// TwinCAT 3 PLC project CycleManagerInterfaceLib
// Title: CNM_CycleManagerInterfaces
// Company: ekvip automation GmbH
// Author: tdie
// ProjectVersion: 0.1.1.0
// Description: A library to provide interfaces and the API for Cycle Managing. .. <legal notes> legal notes ================= | SPDX-FileCopyrightText: © 2024 ekvip automation GmbH <info@ekvip.de> | SPDX-License-Identifier: Apache-2.0 | For details check: Apache-2.0_ .. _Apache-2.0: https://www.apache.org/licenses/LICENSE-2.0 .. </legal notes>
// ProgramVersion: 3.1.4026.19
// libraries:
//   CNM_AbstractObject, * (ekvip automation GmbH)
//   CNM_AssertionInterfaces, * (ekvip automation GmbH)
//   CNM_CommandInterfaces, * (ekvip automation GmbH)
//   CNM_MessageInterfaces, * (ekvip automation GmbH)
//   CNM_ReturnTypes, * (ekvip automation GmbH)
//   Tc2_Standard, * (Beckhoff Automation GmbH)
// project tree:
//   CycleManager/interfaces/configuration/ ICycleManagerConfiguration.TcIO, ICycleManagerConfigurationScope.TcIO, ICycleManagerDefaultParameters.TcIO, ICycleManagerParameters.TcIO, IPauseConfiguration.TcIO, IStopRequestConfiguration.TcIO, ISteppingConfiguration.TcIO, ISequenceConfiguration.TcIO, IStepConfiguration.TcIO, StepStopRequestMode.TcDUT
//   CycleManager/interfaces/ ICycleError.TcIO, ICycleSteps.TcIO
//   CycleManager/SingleExecution/interfaces/ ISingleExecutionCycleManager.TcIO
//   Project Information/ F_GetCompany.TcPOU, F_GetTitle.TcPOU, F_GetVersion.TcPOU
//   Version/ Global_Version.TcGVL
// real-time tasks:
//   TASK PlcTask: cycle T#10ms, priority 20, ADS port 350

// ---- CycleManager/interfaces/configuration/StepStopRequestMode.TcDUT
(*

## Short summary
``StepStopRequestMode`` is an enumeration to control StopRequest behaviour in cycle managers.
Cycle managers should continue with SUCCESS after a stop request is acknowledged by the cycle manager.

.. <legal notes>

legal notes
=================
| SPDX-FileCopyrightText: © 2024 ekvip automation GmbH <info@ekvip.de>
| SPDX-License-Identifier: Apache-2.0
| For details check: Apache-2.0_

.. _Apache-2.0: https://www.apache.org/licenses/LICENSE-2.0

.. </legal notes>

enumeration values
======================

*)

{attribute 'qualified_only'}
{attribute 'strict'}
{attribute 'to_string'}
TYPE StepStopRequestMode :
(
	(*ignore stop request*)
	IGNORE := 0,
	(*proceed with stop request after step finishes and would proceed*)
	AFTER_SUCCESSFUL_STEP := 1,
	(*proceed with stop request only if the step is still busy*)
	ON_BUSY := 2,
	(*immediately proceed with stop request*)
	IMMEDIATE := 3
)DINT;
END_TYPE

// ---- Version/Global_Version.TcGVL
{attribute 'TcGenerated'}
{attribute 'no-analysis'}
{attribute 'linkalways'}
// This function has been automatically generated from the project information.
VAR_GLOBAL CONSTANT
	{attribute 'const_non_replaced'}
	stLibVersion_CNM_CycleManagerInterfaces : ST_LibVersion := (iMajor := 0, iMinor := 1, iBuild := 1, iRevision := 0, nFlags := 0, sVersion := '0.1.1.0');
END_VAR

// ---- CycleManager/interfaces/configuration/ICycleManagerConfiguration.TcIO
(*

## Short summary
An interface to provide configurations for cycle manager in a fluent way.

.. <legal notes>

legal notes
=================
| SPDX-FileCopyrightText: © 2024 ekvip automation GmbH <info@ekvip.de>
| SPDX-License-Identifier: Apache-2.0
| For details check: Apache-2.0_

.. _Apache-2.0: https://www.apache.org/licenses/LICENSE-2.0

.. </legal notes>



*)
INTERFACE ICycleManagerConfiguration EXTENDS __SYSTEM.IQueryInterface

(*

## Short summary
An interface to provide configurations for cycle manager in a fluent way.

.. <legal notes>

legal notes
=================
| SPDX-FileCopyrightText: © 2024 ekvip automation GmbH <info@ekvip.de>
| SPDX-License-Identifier: Apache-2.0
| For details check: Apache-2.0_

.. _Apache-2.0: https://www.apache.org/licenses/LICENSE-2.0

.. </legal notes>



*)
PROPERTY configuration : ICycleManagerConfigurationScope
GET
END_GET
END_PROPERTY

END_INTERFACE

// ---- CycleManager/interfaces/configuration/ICycleManagerConfigurationScope.TcIO
(*

## Short summary
An interface to provide a scope selector for configurations in cycle managers.

.. <legal notes>

legal notes
=================
| SPDX-FileCopyrightText: © 2024 ekvip automation GmbH <info@ekvip.de>
| SPDX-License-Identifier: Apache-2.0
| For details check: Apache-2.0_

.. _Apache-2.0: https://www.apache.org/licenses/LICENSE-2.0

.. </legal notes>



*)
INTERFACE ICycleManagerConfigurationScope EXTENDS __SYSTEM.IQueryInterface

PROPERTY sequence : ISequenceConfiguration
GET
END_GET
END_PROPERTY

PROPERTY step : IStepConfiguration
GET
END_GET
END_PROPERTY

END_INTERFACE

// ---- CycleManager/interfaces/configuration/ICycleManagerDefaultParameters.TcIO
(*

## Short summary
An interface to provide configurations for cycle manager default parameters.
Used internally to allow better fluent implementation.

.. <legal notes>

legal notes
=================
| SPDX-FileCopyrightText: © 2024 ekvip automation GmbH <info@ekvip.de>
| SPDX-License-Identifier: Apache-2.0
| For details check: Apache-2.0_

.. _Apache-2.0: https://www.apache.org/licenses/LICENSE-2.0

.. </legal notes>



*)
INTERFACE ICycleManagerDefaultParameters EXTENDS __System.IQueryInterface

(*

## Short summary
This property sets the default error step for all cycle manager operations.

.. <legal notes>

legal notes
=================
| SPDX-FileCopyrightText: © 2024 ekvip automation GmbH <info@ekvip.de>
| SPDX-License-Identifier: Apache-2.0
| For details check: Apache-2.0_

.. _Apache-2.0: https://www.apache.org/licenses/LICENSE-2.0

.. </legal notes>

*)

PROPERTY defaultErrorStep : DINT
SET
END_SET
END_PROPERTY

(*

## Short summary
This property sets the default pause behavior for all cycle manager operations.

### Usage
This property configures whether pause functionality is enabled by default for the cycle manager.
When enabled, the cycle manager will respond to pause signals and can suspend execution at
appropriate points in the sequence.

The property is write-only and accepts a boolean value to enable or disable pausing.

#### typical usage patterns
1. **Production mode setup**: Enable pausing for production sequences
2. **Maintenance configuration**: Enable pausing for maintenance operations
3. **Automatic operation**: Disable pausing for fully automatic sequences
4. **Operator control**: Enable pausing to allow operator intervention

#### when to use
- During cycle manager initialization to set pause behavior
- When configuring operation modes (automatic vs. manual)
- For setting up operator control capabilities
- When implementing safety or emergency stop procedures

#### behavior details

- When enabled: Cycle manager responds to pause input signals
- When disabled: Pause signals are ignored and sequence continues
- Affects all steps in the sequence unless overridden locally
- Can be overridden on a per-step basis using step configuration

**Example:**
```
// Enable pause for production mode
cyclemanager.configuration.sequence.defaultPauseEnabled := TRUE;

// Disable pause for automatic operation
cyclemanager.configuration.sequence.defaultPauseEnabled := FALSE;

// Configuration based on operation mode
IF operation_mode = OperationMode.MANUAL THEN
	cyclemanager.configuration.sequence.defaultPauseEnabled := TRUE;
ELSE
	cyclemanager.configuration.sequence.defaultPauseEnabled := FALSE;
END_IF;

// Safety configuration
cyclemanager.configuration.sequence
	.defaultPauseEnabled := enable_safety_pause;
```

.. <legal notes>

legal notes
=================
| SPDX-FileCopyrightText: © 2024 ekvip automation GmbH <info@ekvip.de>
| SPDX-License-Identifier: Apache-2.0
| For details check: Apache-2.0_

.. _Apache-2.0: https://www.apache.org/licenses/LICENSE-2.0

.. </legal notes>

*)
PROPERTY defaultPauseEnabled : BOOL
SET
END_SET
END_PROPERTY

(*

## Short summary
Specifies whether the SUCCESS step of the state machine can be skipped when the transition condition to SUCCESS is already fulfilled.

When set to false, the state machine immediately returns SUCCESS as soon as the transition condition to the SUCCESS state is met, 
without executing the dedicated SUCCESS step. This optimization can save one execution cycle per state machine invocation, which is 
especially beneficial in nested or complex state machine structures.

When set to true, the SUCCESS step will always be executed at least once before the state machine returns SUCCESS. This is required 
in cases where the SUCCESS step performs essential actions (e.g., resetting outputs, logging, or cleanup).

The default value is false.

### Use Case:
Use false when the SUCCESS step has no functional side effects and skipping it can improve performance.
Use true when the SUCCESS step contains logic that must be executed explicitly.

.. <legal notes>

legal notes
=================
| SPDX-FileCopyrightText: © 2025 ekvip automation GmbH <info@ekvip.de>
| SPDX-License-Identifier: Apache-2.0
| For details check: Apache-2.0_

.. _Apache-2.0: https://www.apache.org/licenses/LICENSE-2.0

.. </legal notes>

*)

PROPERTY defaultRequireSuccessStep : BOOL
SET
END_SET
END_PROPERTY

(*

## Short summary
This property sets the default stepping mode configuration after a step change.

.. <legal notes>

legal notes
=================
| SPDX-FileCopyrightText: © 2024 ekvip automation GmbH <info@ekvip.de>
| SPDX-License-Identifier: Apache-2.0
| For details check: Apache-2.0_

.. _Apache-2.0: https://www.apache.org/licenses/LICENSE-2.0

.. </legal notes>

*)

PROPERTY defaultSteppingEnabled : BOOL
SET
END_SET
END_PROPERTY

(*

## Short summary
This property sets the default the step width.

.. <legal notes>

legal notes
=================
| SPDX-FileCopyrightText: © 2024 ekvip automation GmbH <info@ekvip.de>
| SPDX-License-Identifier: Apache-2.0
| For details check: Apache-2.0_

.. _Apache-2.0: https://www.apache.org/licenses/LICENSE-2.0

.. </legal notes>

*)

PROPERTY defaultStepWidth : DINT
SET
END_SET
END_PROPERTY

(*

## Short summary
This property sets the default step mode configuration. 

.. <legal notes>

legal notes
=================
| SPDX-FileCopyrightText: © 2024 ekvip automation GmbH <info@ekvip.de>
| SPDX-License-Identifier: Apache-2.0
| For details check: Apache-2.0_

.. _Apache-2.0: https://www.apache.org/licenses/LICENSE-2.0

.. </legal notes>

*)

PROPERTY defaultStopRequestMode :StepStopRequestMode
SET
END_SET
END_PROPERTY

(*

## Short summary
This property sets the maximum execution time for steps. 
The cycle manager will go into the timeoutStep after the time elapsed.

.. <legal notes>

legal notes
=================
| SPDX-FileCopyrightText: © 2024 ekvip automation GmbH <info@ekvip.de>
| SPDX-License-Identifier: Apache-2.0
| For details check: Apache-2.0_

.. _Apache-2.0: https://www.apache.org/licenses/LICENSE-2.0

.. </legal notes>

*)

PROPERTY defaultTimeout : TIME
SET
END_SET
END_PROPERTY

(*

## Short summary
This property sets the default step that will be set if the current step reaches a timeout. 

.. <legal notes>

legal notes
=================
| SPDX-FileCopyrightText: © 2024 ekvip automation GmbH <info@ekvip.de>
| SPDX-License-Identifier: Apache-2.0
| For details check: Apache-2.0_

.. _Apache-2.0: https://www.apache.org/licenses/LICENSE-2.0

.. </legal notes>

*)

PROPERTY defaultTimeoutStep : DINT
SET
END_SET
END_PROPERTY

END_INTERFACE

// ---- CycleManager/interfaces/configuration/ICycleManagerParameters.TcIO
(*

## Short summary
An interface to provide configurations for the cycle manager parameters.

.. <legal notes>

legal notes
=================
| SPDX-FileCopyrightText: © 2024 ekvip automation GmbH <info@ekvip.de>
| SPDX-License-Identifier: Apache-2.0
| For details check: Apache-2.0_

.. _Apache-2.0: https://www.apache.org/licenses/LICENSE-2.0

.. </legal notes>



*)
INTERFACE ICycleManagerParameters EXTENDS __System.IQueryInterface

(*

## Short summary
This property sets the next step in case of an error.

.. <legal notes>

legal notes
=================
| SPDX-FileCopyrightText: © 2024 ekvip automation GmbH <info@ekvip.de>
| SPDX-License-Identifier: Apache-2.0
| For details check: Apache-2.0_

.. _Apache-2.0: https://www.apache.org/licenses/LICENSE-2.0

.. </legal notes>

*)
PROPERTY errorStep :DINT
SET
END_SET
END_PROPERTY

(*

## Short summary
This property allows enabling and disabling pausing.

.. <legal notes>

legal notes
=================
| SPDX-FileCopyrightText: © 2024 ekvip automation GmbH <info@ekvip.de>
| SPDX-License-Identifier: Apache-2.0
| For details check: Apache-2.0_

.. _Apache-2.0: https://www.apache.org/licenses/LICENSE-2.0

.. </legal notes>

*)

PROPERTY pause : IPauseConfiguration
GET
END_GET
END_PROPERTY

(*

## Short summary
This property allows enabling and disabling stepping mode.

.. <legal notes>

legal notes
=================
| SPDX-FileCopyrightText: © 2024 ekvip automation GmbH <info@ekvip.de>
| SPDX-License-Identifier: Apache-2.0
| For details check: Apache-2.0_

.. _Apache-2.0: https://www.apache.org/licenses/LICENSE-2.0

.. </legal notes>

*)

PROPERTY stepping : ISteppingConfiguration
GET
END_GET
END_PROPERTY

(*

## Short summary
This property sets the step width when proceeding automatically.
This defaults to 1.

.. <legal notes>

legal notes
=================
| SPDX-FileCopyrightText: © 2024 ekvip automation GmbH <info@ekvip.de>
| SPDX-License-Identifier: Apache-2.0
| For details check: Apache-2.0_

.. _Apache-2.0: https://www.apache.org/licenses/LICENSE-2.0

.. </legal notes>

*)
PROPERTY stepWidth : DINT
SET
END_SET
END_PROPERTY

(*

## Short summary
This property allows changing the stop request behaviour in case of active stop request.

.. <legal notes>

legal notes
=================
| SPDX-FileCopyrightText: © 2024 ekvip automation GmbH <info@ekvip.de>
| SPDX-License-Identifier: Apache-2.0
| For details check: Apache-2.0_

.. _Apache-2.0: https://www.apache.org/licenses/LICENSE-2.0

.. </legal notes>

*)
PROPERTY stopRequest : IStopRequestConfiguration
GET
END_GET
END_PROPERTY

(*

## Short summary
This property sets the maximum execution time for steps. 
The cycle manager will go into the timeoutStep after the time elapsed.
Set to T#0MS for no timeout (infinite), default.

.. <legal notes>

legal notes
=================
| SPDX-FileCopyrightText: © 2024 ekvip automation GmbH <info@ekvip.de>
| SPDX-License-Identifier: Apache-2.0
| For details check: Apache-2.0_

.. _Apache-2.0: https://www.apache.org/licenses/LICENSE-2.0

.. </legal notes>

*)
PROPERTY timeout :TIME
SET
END_SET
END_PROPERTY

(*

## Short summary
This property sets the step that will be set if the current step reaches a timeout. 
If not changed will default to the current errorStep.

.. <legal notes>

legal notes
=================
| SPDX-FileCopyrightText: © 2024 ekvip automation GmbH <info@ekvip.de>
| SPDX-License-Identifier: Apache-2.0
| For details check: Apache-2.0_

.. _Apache-2.0: https://www.apache.org/licenses/LICENSE-2.0

.. </legal notes>

*)
PROPERTY timeoutStep :DINT
SET
END_SET
END_PROPERTY

END_INTERFACE

// ---- CycleManager/interfaces/configuration/IPauseConfiguration.TcIO
(*

## Short summary
An interface to enable and diable pause functionallity.

.. <legal notes>

legal notes
=================
| SPDX-FileCopyrightText: © 2024 ekvip automation GmbH <info@ekvip.de>
| SPDX-License-Identifier: Apache-2.0
| For details check: Apache-2.0_

.. _Apache-2.0: https://www.apache.org/licenses/LICENSE-2.0

.. </legal notes>



*)
INTERFACE IPauseConfiguration EXTENDS __System.IQueryInterface

(*

## Short summary
This method disables pausing, disabling the cycle manager transition to PAUSED even if pause signal is active.

.. <legal notes>

legal notes
=================
| SPDX-FileCopyrightText: © 2024 ekvip automation GmbH <info@ekvip.de>
| SPDX-License-Identifier: Apache-2.0
| For details check: Apache-2.0_

.. _Apache-2.0: https://www.apache.org/licenses/LICENSE-2.0

.. </legal notes>

*)
METHOD disable
END_METHOD

(*

## Short summary
This method enables pausing, allowing the cycle manager to transition to PAUSED state if pause is active.

.. <legal notes>

legal notes
=================
| SPDX-FileCopyrightText: © 2024 ekvip automation GmbH <info@ekvip.de>
| SPDX-License-Identifier: Apache-2.0
| For details check: Apache-2.0_

.. _Apache-2.0: https://www.apache.org/licenses/LICENSE-2.0

.. </legal notes>

*)

METHOD enable
END_METHOD

END_INTERFACE

// ---- CycleManager/interfaces/configuration/IStopRequestConfiguration.TcIO
(*

## Short summary
An interface to configure stop request behavior.

.. <legal notes>

legal notes
=================
| SPDX-FileCopyrightText: © 2024 ekvip automation GmbH <info@ekvip.de>
| SPDX-License-Identifier: Apache-2.0
| For details check: Apache-2.0_

.. _Apache-2.0: https://www.apache.org/licenses/LICENSE-2.0

.. </legal notes>



*)
INTERFACE IStopRequestConfiguration EXTENDS __System.IQueryInterface

(*

## Short summary
This method sets the stop request behaviour to ``StepStopRequestMode.AFTER_SUCCESSFUL_STEP``.
If the StopRequest signal is active, the cycle manager will move to succees if the current step was successful during the update call.

.. <legal notes>

legal notes
=================
| SPDX-FileCopyrightText: © 2024 ekvip automation GmbH <info@ekvip.de>
| SPDX-License-Identifier: Apache-2.0
| For details check: Apache-2.0_

.. _Apache-2.0: https://www.apache.org/licenses/LICENSE-2.0

.. </legal notes>


*)

METHOD afterSuccessfulStep
END_METHOD

(*

## Short summary
This method sets the stop request behaviour to ``StepStopRequestMode.IGNORE``.
The cycle manager will ignore the stop request signal.

.. <legal notes>

legal notes
=================
| SPDX-FileCopyrightText: © 2024 ekvip automation GmbH <info@ekvip.de>
| SPDX-License-Identifier: Apache-2.0
| For details check: Apache-2.0_

.. _Apache-2.0: https://www.apache.org/licenses/LICENSE-2.0

.. </legal notes>


*)

METHOD ignore
END_METHOD

(*

## Short summary
This method sets the stop request behaviour to ``StepStopRequestMode.IMMEDIATE``.
If the StopRequest signal is active, the cycle manager will always move to succees during the update call.

.. <legal notes>

legal notes
=================
| SPDX-FileCopyrightText: © 2024 ekvip automation GmbH <info@ekvip.de>
| SPDX-License-Identifier: Apache-2.0
| For details check: Apache-2.0_

.. _Apache-2.0: https://www.apache.org/licenses/LICENSE-2.0

.. </legal notes>


*)

METHOD immediate
END_METHOD

(*

## Short summary
This method sets the stop request behaviour to ``StepStopRequestMode.ON_BUSY``.
If the StopRequest signal is active, the cycle manager will move to succees if the current step was busy during the update call.

.. <legal notes>

legal notes
=================
| SPDX-FileCopyrightText: © 2024 ekvip automation GmbH <info@ekvip.de>
| SPDX-License-Identifier: Apache-2.0
| For details check: Apache-2.0_

.. _Apache-2.0: https://www.apache.org/licenses/LICENSE-2.0

.. </legal notes>

*)

METHOD onBusy
END_METHOD

END_INTERFACE

// ---- CycleManager/interfaces/configuration/ISteppingConfiguration.TcIO
(*

## Short summary
An interface to provide stepping behaviour to cycle managers.

.. <legal notes>

legal notes
=================
| SPDX-FileCopyrightText: © 2024 ekvip automation GmbH <info@ekvip.de>
| SPDX-License-Identifier: Apache-2.0
| For details check: Apache-2.0_

.. _Apache-2.0: https://www.apache.org/licenses/LICENSE-2.0

.. </legal notes>



*)
INTERFACE ISteppingConfiguration EXTENDS __System.IQueryInterface

(*

## Short summary
This method disables step mode, allowing automatic proceeding without using the step signal.

.. <legal notes>

legal notes
=================
| SPDX-FileCopyrightText: © 2024 ekvip automation GmbH <info@ekvip.de>
| SPDX-License-Identifier: Apache-2.0
| For details check: Apache-2.0_

.. _Apache-2.0: https://www.apache.org/licenses/LICENSE-2.0

.. </legal notes>

*)
METHOD disable
END_METHOD

(*

## Short summary
This method enables step mode, only allowing automatic proceeding if the step signal is active.

.. <legal notes>

legal notes
=================
| SPDX-FileCopyrightText: © 2024 ekvip automation GmbH <info@ekvip.de>
| SPDX-License-Identifier: Apache-2.0
| For details check: Apache-2.0_

.. _Apache-2.0: https://www.apache.org/licenses/LICENSE-2.0

.. </legal notes>

*)
METHOD enable
END_METHOD

END_INTERFACE

// ---- CycleManager/interfaces/configuration/ISequenceConfiguration.TcIO
(*

## Short summary
An interface to provide configurations for all cycle manager steps.
Should affect the all steps in the cycle manager (default values).

.. <legal notes>

legal notes
=================
| SPDX-FileCopyrightText: © 2024 ekvip automation GmbH <info@ekvip.de>
| SPDX-License-Identifier: Apache-2.0
| For details check: Apache-2.0_

.. _Apache-2.0: https://www.apache.org/licenses/LICENSE-2.0

.. </legal notes>



*)
INTERFACE ISequenceConfiguration EXTENDS ICycleManagerParameters

(*

## Short summary
Specifies whether the SUCCESS step of the state machine can be skipped when the transition condition to SUCCESS is already fulfilled.

When set to false, the state machine immediately returns SUCCESS as soon as the transition condition to the SUCCESS state is met, 
without executing the dedicated SUCCESS step. This optimization can save one execution cycle per state machine invocation, which is 
especially beneficial in nested or complex state machine structures.

When set to true, the SUCCESS step will always be executed at least once before the state machine returns SUCCESS. This is required 
in cases where the SUCCESS step performs essential actions (e.g., resetting outputs, logging, or cleanup).

The default value is false.

### Use Case
Use false when the SUCCESS step has no functional side effects and skipping it can improve performance.
Use true when the SUCCESS step contains logic that must be executed explicitly.

.. <legal notes>

legal notes
=================
| SPDX-FileCopyrightText: © 2025 ekvip automation GmbH <info@ekvip.de>
| SPDX-License-Identifier: Apache-2.0
| For details check: Apache-2.0_

.. _Apache-2.0: https://www.apache.org/licenses/LICENSE-2.0

.. </legal notes>

*)

PROPERTY requireSuccessStep : BOOL
SET
END_SET
END_PROPERTY

END_INTERFACE

// ---- CycleManager/interfaces/configuration/IStepConfiguration.TcIO
(*

## Short summary
An interface to provide configurations for cycle manager steps.
Should only affect the currently active step.

.. <legal notes>

legal notes
=================
| SPDX-FileCopyrightText: © 2024 ekvip automation GmbH <info@ekvip.de>
| SPDX-License-Identifier: Apache-2.0
| For details check: Apache-2.0_

.. _Apache-2.0: https://www.apache.org/licenses/LICENSE-2.0

.. </legal notes>



*)
INTERFACE IStepConfiguration EXTENDS ICycleManagerParameters

END_INTERFACE

// ---- CycleManager/interfaces/ICycleError.TcIO
(*

## Short summary
An interface to provide error handling in cycle management.

.. <legal notes>

legal notes
=================
| SPDX-FileCopyrightText: © 2024 ekvip automation GmbH <info@ekvip.de>
| SPDX-License-Identifier: Apache-2.0
| For details check: Apache-2.0_

.. _Apache-2.0: https://www.apache.org/licenses/LICENSE-2.0

.. </legal notes>



*)
INTERFACE ICycleError EXTENDS __System.IQueryInterface

(*

## Short summary
This method acknowledges an error in the cycle manager 
and resets the current step to the step before the error occurred.


### Purpose and usage
This method provides error acknowledgment functionality for the cycle manager. It clears the current error state
and returns the cycle manager to the step that was executing before the error occurred, allowing for error recovery
and continuation of the sequence.

The method should be called when an operator or system wants to acknowledge an error and attempt to continue
the process from where it left off.

### Typical usage patterns

1. **Manual error acknowledgment**: Operator acknowledges error via HMI button
2. **Automatic error recovery**: System automatically acknowledges after conditions are met
3. **Retry operations**: Acknowledge error to retry the failed step
4. **Error logging**: Acknowledge error after logging for audit trail

#### When to use

- When an error has been resolved and process should continue
- After manual operator intervention to fix the error condition
- In automated error recovery scenarios
- When implementing retry logic after temporary failures

### behavior

- Clears the error state flag
- Returns cycle manager to the last successful step
- Resets internal error tracking variables
- Allows normal sequence progression to resume

**Example:**
```
// Manual error acknowledgment via HMI
IF HMI_acknowledge_button THEN
	cyclemanager.errors.acknowledge();
	HMI_acknowledge_button := FALSE;
END_IF;

// Automatic error acknowledgment after condition resolution
ERROR_STEP:
	IF error_condition_resolved THEN
		cyclemanager.errors.acknowledge();  // Return to previous step
	END_IF;

// Error acknowledgment with logging
IF error_acknowledged_by_operator THEN
	logger.logEvent('Error acknowledged by operator');
	cyclemanager.errors.acknowledge();
	error_acknowledged_by_operator := FALSE;
END_IF;
```

.. <legal notes>

legal notes
=================
| SPDX-FileCopyrightText: © 2024 ekvip automation GmbH <info@ekvip.de>
| SPDX-License-Identifier: Apache-2.0
| For details check: Apache-2.0_

.. _Apache-2.0: https://www.apache.org/licenses/LICENSE-2.0

.. </legal notes>

*)
METHOD acknowledge
END_METHOD

(*

## Short summary
This method throws an alarm and waits for it to be confirmed. 
When the alarm was confirmed the cyclemanager will proceed to next configured step.
If the current step is the result of an evaluated error state and the input 'resumeWithLastStep' is set to true, the cyclemanager will proceed to the last step.
**Warning:**  The 'resumeWithLastStep' flag will be ignored if the last step was successful.

### Purpose and usage
This method provides comprehensive error handling by displaying an alarm to the operator and managing 
the subsequent cycle manager behavior based on the error acknowledgment. It integrates alarm management
with cycle flow control for robust error handling.

The method blocks execution until the alarm is acknowledged and then determines the next step based
on the error context and resumeWithLastStep parameter.

### Typical usage patterns
1. **Critical error handling**: Display alarm for critical errors requiring operator intervention
2. **Process deviation handling**: Show alarm when process parameters are out of range
3. **Equipment failure handling**: Alert operators to equipment malfunctions
4. **Recovery operations**: Provide options for continuing after error resolution

### When to use
- When an error requires operator notification and acknowledgment
- For errors that need to be logged and tracked in the alarm system
- When you need flexible recovery options (continue or retry)
- For integrating cycle management with plant-wide alarm systems

### Behaviour details
- Displays the alarm using the CNM message system
- Blocks cycle progression until alarm is acknowledged
- If resumeWithLastStep=TRUE and step was reached via error: returns to last step
- If resumeWithLastStep=FALSE: proceeds to next configured step
- Warning: resumeWithLastStep is ignored if last step was successful

### Parameter validation
- alarm parameter must be a valid IAlarm instance
- resumeWithLastStep flag only affects behavior when current step resulted from error evaluation

**Example:**
```
// Basic error handling with alarm
PROCESS_STEP:
	IF motor_overload_detected THEN
		cyclemanager.errors.handle(motor_overload_alarm, TRUE);  // Resume with last step after ack
	END_IF;

// Error handling with different recovery strategies
CRITICAL_OPERATION:
	IF safety_violation THEN
		cyclemanager.errors.handle(safety_alarm, FALSE);  // Don't resume, go to next step
	ELSIF equipment_fault THEN
		cyclemanager.errors.handle(equipment_alarm, TRUE);  // Allow retry of operation
	END_IF;

// Complex error handling with context
VAR
	process_error_alarm : ProcessErrorAlarm;
END_VAR

MONITORING_STEP:
	IF temperature_out_of_range THEN
		process_error_alarm.setMessage('Temperature exceeded limits');
		process_error_alarm.setSeverity(AlarmSeverity.WARNING);
		cyclemanager.errors.handle(process_error_alarm, TRUE);
	END_IF;
```

.. <legal notes>

legal notes
=================
| SPDX-FileCopyrightText: © 2024 ekvip automation GmbH <info@ekvip.de>
| SPDX-License-Identifier: Apache-2.0
| For details check: Apache-2.0_

.. _Apache-2.0: https://www.apache.org/licenses/LICENSE-2.0

.. </legal notes>

*)

METHOD handle
VAR_INPUT
	(* the alarm event that should be thrown *)
	alarm :CNM_MessageInterfaces.IAlarm;
	(* if this flag is set AND we got to the current step because of an ERROR state, then the cyclemanager will automatically will go back to the last step *)
	resumeWithLastStep :BOOL := TRUE;
END_VAR
END_METHOD

(*

## Short summary
This property returns TRUE if the step was reached by evaluating an error.

### Purpose and usage
This property provides status information about how the current step was reached. It indicates whether 
the cycle manager arrived at the current step as a result of an error evaluation, which is crucial
for implementing context-aware error handling and recovery logic.

The property is read-only and returns a boolean value indicating error context.

**return**
BOOL: TRUE if current step was reached by error evaluation, FALSE if reached through normal flow

### Typical usage patterns
1. **Conditional error handling**: Different behavior based on how step was reached
2. **Recovery decision making**: Determine appropriate recovery actions
3. **Error logging**: Log additional context about error conditions
4. **UI feedback**: Show different information based on error context

### When to use
- In error handling steps to determine recovery strategy
- When implementing different behaviors for error vs. normal flow
- For logging and audit trail purposes
- In HMI displays to show appropriate error context

### Behaviour details
- Returns TRUE when step was reached via error evaluation (e.g., command returned ERROR state)
- Returns FALSE when step was reached through normal progression
- Useful for implementing smart error recovery logic
- Context is maintained until step changes or error is acknowledged

**Example:**
```
// Context-aware error handling
ERROR_STEP:
	IF cyclemanager.errors.isInErrorStep THEN
		// This step was reached due to an error
		display_error_message := 'Process failed - manual intervention required';
		allow_retry := TRUE;
	ELSE
		// This step was reached through normal flow
		display_error_message := 'Manual error step - check process conditions';
		allow_retry := FALSE;
	END_IF;

// Different recovery strategies based on context
RECOVERY_STEP:
	IF cyclemanager.errors.isInErrorStep THEN
		// Automatic retry for error-triggered steps
		IF retry_count < MAX_RETRIES THEN
			cyclemanager.errors.acknowledge();  // Try again
		ELSE
			cyclemanager.steps.next := ABORT_STEP;  // Give up
		END_IF;
	ELSE
		// Manual step - wait for operator decision
		cyclemanager.waitFor(operator_continue_signal);
	END_IF;

// Error logging with context
IF log_step_entry THEN
	IF cyclemanager.errors.isInErrorStep THEN
		logger.logError('Entered step due to error condition');
	ELSE
		logger.logInfo('Entered step through normal flow');
	END_IF;
	log_step_entry := FALSE;
END_IF;

.. <legal notes>

legal notes
=================
| SPDX-FileCopyrightText: © 2024 ekvip automation GmbH <info@ekvip.de>
| SPDX-License-Identifier: Apache-2.0
| For details check: Apache-2.0_

.. _Apache-2.0: https://www.apache.org/licenses/LICENSE-2.0

.. </legal notes>

*)
PROPERTY isInErrorStep : BOOL
GET
END_GET
END_PROPERTY

END_INTERFACE

// ---- CycleManager/interfaces/ICycleSteps.TcIO
(*

## Short summary
An interface to provide last, current and next step properties in cycle management.

.. <legal notes>

legal notes
=================
| SPDX-FileCopyrightText: © 2024 ekvip automation GmbH <info@ekvip.de>
| SPDX-License-Identifier: Apache-2.0
| For details check: Apache-2.0_

.. _Apache-2.0: https://www.apache.org/licenses/LICENSE-2.0

.. </legal notes>



*)
INTERFACE ICycleSteps EXTENDS __System.IQueryInterface

(*

## Short summary
This property returns the current step of the cycle manager.
Proposed use is as CASE control.

### Purpose and usage
This property provides the current step number of the cycle manager for implementing step-based control logic.
It is primarily used in CASE statements to execute different actions based on the current step.

The property is read-only and returns the current step as a DINT value.

**return**
DINT: Current step number of the cycle manager

### Typical usage patterns
1. **CASE control structure**: Main usage in CASE statements for step-based execution
2. **Step monitoring**: Reading current step for HMI display or logging
3. **Conditional logic**: Checking current step for specific conditions

### When to use
- In every cycle manager implementation for step-based control
- When you need to display current step status
- For debugging and logging purposes
- When implementing conditional logic based on current step

**Example:**
```
CASE cyclemanager.steps.current OF
DefaultSteps.STEP.IDLE:
	// Initialize sequence
	;
DefaultSteps.STEP.INIT:
	// Perform initialization
	;
2:
	// Custom step - move to position
	;
3:
	// Custom step - perform operation
	;
4:
	// Custom step - finalize
	;
DefaultSteps.STEP.SUCCESS:
	// Sequence completed successfully
	;
DefaultSteps.STEP.ERROR:
	// Handle error conditions
	;
DefaultSteps.STEP.ABORT:
	// Handle abort conditions
	;
ELSE 
	// Handle unexpected steps
	;
END_CASE

// Usage for monitoring
currentStepForHMI := cyclemanager.steps.current;
```

.. <legal notes>

legal notes
=================
| SPDX-FileCopyrightText: © 2024 ekvip automation GmbH <info@ekvip.de>
| SPDX-License-Identifier: Apache-2.0
| For details check: Apache-2.0_

.. _Apache-2.0: https://www.apache.org/licenses/LICENSE-2.0

.. </legal notes>

*)
PROPERTY current :DINT
GET
END_GET
END_PROPERTY

(*

## Short summary
This property returns the last step of the cycle manager, useful for error steps.

### Purpose and usage
This property provides the last executed step number of the cycle manager, primarily used for error handling and recovery operations.
It allows returning to the previous step for retry operations or error recovery procedures.

The property is read-only and returns the last step as a DINT value.

**return**
DINT: Last executed step number of the cycle manager

### Typical usage patterns
1. **Error recovery**: Returning to previous step after error handling
2. **Retry operations**: Going back one step to retry failed operations
3. **Step debugging**: Tracking step transitions for debugging purposes
4. **Conditional branching**: Making decisions based on where the error occurred

### When to use
- In error handling steps to implement retry logic
- When you need to return to the previous step after error resolution
- For debugging step transitions and sequence flow
- In timeout handling to retry the previous operation

**Example:**
```
// Error handling with retry logic
TIMEOUT_STEP_FOR_RETRY:
	cM.steps.next := cM.steps.last - 1;  // Go back to previous step
	cM.waitFor(ACK);

// Error step with conditional recovery
DefaultSteps.STEP.ERROR:
	IF retry_counter < MAX_RETRIES THEN
		retry_counter := retry_counter + 1;
		cM.steps.next := cM.steps.last;  // Retry the failed step
	ELSE
		cM.steps.next := DefaultSteps.STEP.ABORT;  // Give up after max retries
	END_IF;

// Step transition logging
logger.logStepTransition(cM.steps.last, cM.steps.current);
```

.. <legal notes>

legal notes
=================
| SPDX-FileCopyrightText: © 2024 ekvip automation GmbH <info@ekvip.de>
| SPDX-License-Identifier: Apache-2.0
| For details check: Apache-2.0_

.. _Apache-2.0: https://www.apache.org/licenses/LICENSE-2.0

.. </legal notes>

*)
PROPERTY last :DINT
GET
END_GET
END_PROPERTY

(*

## Short summary
This property sets the next step of the cycle manager.

### Purpose and usage
This property sets the next step that the cycle manager should execute after completing the current step.
It provides explicit control over the sequence flow, allowing for conditional branching, error handling, and custom step sequencing.

The property is write-only and accepts a DINT value representing the target step number.

### Typical usage patterns
1. **Conditional branching**: Setting different next steps based on conditions
2. **Error handling**: Directing flow to error or recovery steps
3. **Sequential control**: Explicitly controlling step progression
4. **Skip operations**: Jumping over steps that are not needed

### When to use
- When you need to control step progression explicitly
- For conditional branching based on process conditions
- In error handling to redirect to error steps
- When implementing complex sequence logic with jumps
- For skipping steps that are not required in current context

### Parameter validation
- Step number should be a valid step in your sequence
- Negative step numbers are typically reserved for system steps
- Use DefaultSteps.STEP constants for standard steps (IDLE, INIT, SUCCESS, ERROR, ABORT)

**Example:**
```
// Conditional branching
MY_STEP:
	IF process_complete THEN
		cyclemanager.steps.next := SUCCESS_STEP;
	ELSE
		cyclemanager.steps.next := CONTINUE_PROCESS_STEP;
	END_IF;
	cyclemanager.executeCommand(finalizeProcess);

// Error handling
PROCESS_STEP:
	IF error_detected THEN
		cyclemanager.steps.next := DefaultSteps.STEP.ERROR;
	ELSE
		cyclemanager.steps.next := NEXT_PROCESS_STEP;
	END_IF;

// Skip operation based on condition
OPTIONAL_STEP_CHECK:
	IF skip_calibration THEN
		cyclemanager.steps.next := MAIN_OPERATION_STEP;  // Skip calibration
	ELSE
		cyclemanager.steps.next := CALIBRATION_STEP;     // Perform calibration
	END_IF;
```

.. <legal notes>

legal notes
=================
| SPDX-FileCopyrightText: © 2024 ekvip automation GmbH <info@ekvip.de>
| SPDX-License-Identifier: Apache-2.0
| For details check: Apache-2.0_

.. _Apache-2.0: https://www.apache.org/licenses/LICENSE-2.0

.. </legal notes>

*)
PROPERTY next :DINT
GET
END_GET
SET
END_SET
END_PROPERTY

END_INTERFACE

// ---- CycleManager/SingleExecution/interfaces/ISingleExecutionCycleManager.TcIO
(*

## Short summary
An interface to provide simple cycle management for steps in state machines.

.. <legal notes>

legal notes
=================
| SPDX-FileCopyrightText: © 2024 ekvip automation GmbH <info@ekvip.de>
| SPDX-License-Identifier: Apache-2.0
| For details check: Apache-2.0_

.. _Apache-2.0: https://www.apache.org/licenses/LICENSE-2.0

.. </legal notes>



*)
INTERFACE ISingleExecutionCycleManager 
EXTENDS CNM_AbstractObject.IObject, 
	CNM_AssertionInterfaces.IAssertor, 
	ICycleError, 
	ICycleSteps, 
	ICycleManagerConfiguration

(*

## Short summary
This method performs the given invoke only in the first cycle of the current step.

### Purpose and usage
This method provides step entry functionality for the cycle manager. It executes a single-attempt command
only on the first cycle when entering a step, making it ideal for initialization operations, setting outputs,
or triggering one-time actions at the beginning of a step.

The method ensures the command is executed exactly once per step entry, regardless of how many cycles
the step remains active.


### Typical usage patterns
1. **Step initialization**: Setting up conditions when entering a step
2. **Output control**: Activating outputs or devices at step start
3. **Data logging**: Recording step entry events
4. **Communication**: Sending messages or signals on step entry

### When to use
- When you need one-time execution at the beginning of a step
- For initializing variables or conditions when entering a step
- When activating outputs that should remain active during the step
- For triggering events that should only happen once per step entry

### Behaviour details
- Command is executed only in the first cycle of the current step
- Subsequent cycles in the same step do not re-execute the command
- If command fails, cycle manager proceeds to specified errorStep
- If command succeeds, normal step progression continues

### Parameter validation
- invoke must be a valid ISingleAttempt command instance
- errorStep should be a valid step number (typically negative for system steps)

**Example:**
```
// Initialize outputs when entering step
STEP_START_CONVEYOR:
	cyclemanager.enter(activateConveyorCommand, CONVEYOR_ERROR_STEP);
	cyclemanager.proceed();

// Set variables on step entry
STEP_PREPARE_OPERATION:
	cyclemanager.enter(setOperationParametersCommand);
	cyclemanager.waitFor(parameters_ready);

// Trigger communication on step entry
STEP_NOTIFY_MES:
	cyclemanager.enter(sendMESUpdateCommand, COMMUNICATION_ERROR_STEP);
	cyclemanager.proceed();

// Complex step with multiple entry actions
STEP_COMPLEX_INIT:
	cyclemanager.enter(initializeSystemCommand);
	IF cyclemanager.executeStep THEN
		// Additional logic after first cycle
		monitor_initialization_progress();
	END_IF;
	cyclemanager.waitFor(initialization_complete);

```

.. <legal notes>

legal notes
=================
| SPDX-FileCopyrightText: © 2024 ekvip automation GmbH <info@ekvip.de>
| SPDX-License-Identifier: Apache-2.0
| For details check: Apache-2.0_

.. _Apache-2.0: https://www.apache.org/licenses/LICENSE-2.0

.. </legal notes>

*)

METHOD enter
VAR_INPUT
	(* command to execute *)
	invoke :CNM_CommandInterfaces.ISingleAttempt;
	(* step to proceed with in case of error *)
	errorStep :DINT := CNM_ReturnTypes.DefaultSteps.STEP.ERROR;
END_VAR
END_METHOD

(*

## Short summary
This property returns an ``ICycleError`` interface fluently to provide error handling methods.

### Purpose and usage
This property provides fluent access to the error handling interface of the cycle manager. It allows
chaining error-related method calls and enables comprehensive error management functionality within
the cycle management system.

The property returns the same instance cast to ICycleError interface for method chaining.

**return:** 
ICycleError: Error handling interface providing acknowledge() and handle() methods

### Typical usage patterns
1. **Fluent error acknowledgment**: Chain method calls for cleaner code
2. **Error handling**: Access error-specific methods and properties
3. **Error state checking**: Check if current step was reached via error
4. **Alarm integration**: Handle errors with alarm system integration

### When to use
- When you need to acknowledge errors in the cycle
- For displaying alarms and waiting for operator response
- When implementing error recovery logic
- For fluent method chaining in error scenarios

**Example:**
```
// Fluent error acknowledgment
IF operator_ack_button THEN
	cyclemanager.errors.acknowledge();
END_IF;

// Error handling with alarm
IF critical_error_detected THEN
	cyclemanager.errors.handle(critical_alarm, TRUE);
END_IF;

// Check error context
IF cyclemanager.errors.isInErrorStep THEN
	// Handle error-triggered step differently
	enable_manual_mode := TRUE;
ELSE
	enable_manual_mode := FALSE;
END_IF;

// Fluent chaining (conceptual - methods don't return interfaces)
// This demonstrates the fluent interface pattern
error_interface := cyclemanager.errors;
error_interface.acknowledge();
```

.. <legal notes>

legal notes
=================
| SPDX-FileCopyrightText: © 2024 ekvip automation GmbH <info@ekvip.de>
| SPDX-License-Identifier: Apache-2.0
| For details check: Apache-2.0_

.. _Apache-2.0: https://www.apache.org/licenses/LICENSE-2.0

.. </legal notes>

*)
PROPERTY errors :ICycleError
GET
END_GET
END_PROPERTY

(*

## Short summary
This method evaluates an execution state to calculate the next step.

.. <legal notes>

legal notes
=================
| SPDX-FileCopyrightText: © 2024 ekvip automation GmbH <info@ekvip.de>
| SPDX-License-Identifier: Apache-2.0
| For details check: Apache-2.0_

.. _Apache-2.0: https://www.apache.org/licenses/LICENSE-2.0

.. </legal notes>

*)
METHOD evaluate
VAR_INPUT
	(* the state which is to be evaluated *)
	state :CNM_ReturnTypes.SingleExecutionState;
	(* step to proceed with in case of error *)
	errorStep :DINT := CNM_ReturnTypes.DefaultSteps.STEP.ERROR;
END_VAR
END_METHOD

(*

## Short summary
This method performs the given command and evaluates the return value.
The command will be called with execute := FALSE in the first cycle and with execute := TRUE in all following

.. <legal notes>

legal notes
=================
| SPDX-FileCopyrightText: © 2024 ekvip automation GmbH <info@ekvip.de>
| SPDX-License-Identifier: Apache-2.0
| For details check: Apache-2.0_

.. _Apache-2.0: https://www.apache.org/licenses/LICENSE-2.0

.. </legal notes>

*)
METHOD executeCommand
VAR_INPUT
	(* command to execute *)
	command :CNM_CommandInterfaces.ICommand;
	(* step to proceed with in case of error *)
	errorStep :DINT := CNM_ReturnTypes.DefaultSteps.STEP.ERROR;
END_VAR
END_METHOD

(*

## Short summary
This property returns the execute flag for the current step, 
which is FALSE in the first cycle of each step and TRUE after.

.. <legal notes>

legal notes
=================
| SPDX-FileCopyrightText: © 2024 ekvip automation GmbH <info@ekvip.de>
| SPDX-License-Identifier: Apache-2.0
| For details check: Apache-2.0_

.. _Apache-2.0: https://www.apache.org/licenses/LICENSE-2.0

.. </legal notes>

*)
PROPERTY executeStep :BOOL
GET
END_GET
END_PROPERTY

(*

## Short summary
This method performs the given invoke only in the last cycle of the current step.

.. <legal notes>

legal notes
=================
| SPDX-FileCopyrightText: © 2024 ekvip automation GmbH <info@ekvip.de>
| SPDX-License-Identifier: Apache-2.0
| For details check: Apache-2.0_

.. _Apache-2.0: https://www.apache.org/licenses/LICENSE-2.0

.. </legal notes>

*)
METHOD leave
VAR_INPUT
	(* command to execute *)
	invoke :CNM_CommandInterfaces.ISingleAttempt;
	(* step to proceed with in case of error *)
	errorStep :DINT := CNM_ReturnTypes.DefaultSteps.STEP.ERROR;
	(* whether the attempt should be called even if there was an error in the current step *)
	forceOnError :BOOL := FALSE;
END_VAR
END_METHOD

(*

## Short summary
This method changes the current step in the cycle manager to the next in order (current + stepWidth) .
If any evaluate or other call is still busy it will ignore them and change to the next step.

.. <legal notes>

legal notes
=================
| SPDX-FileCopyrightText: © 2024 ekvip automation GmbH <info@ekvip.de>
| SPDX-License-Identifier: Apache-2.0
| For details check: Apache-2.0_

.. _Apache-2.0: https://www.apache.org/licenses/LICENSE-2.0

.. </legal notes>

*)
METHOD proceed
END_METHOD

(*

## Short summary
This method changes the current step in the cycle manager to the given step.
If any evaluate or other call is still busy it will ignore them and move to the next step.

.. <legal notes>

legal notes
=================
| SPDX-FileCopyrightText: © 2024 ekvip automation GmbH <info@ekvip.de>
| SPDX-License-Identifier: Apache-2.0
| For details check: Apache-2.0_

.. _Apache-2.0: https://www.apache.org/licenses/LICENSE-2.0

.. </legal notes>

*)
METHOD proceedWith
VAR_INPUT
	(* step to move to *)
	step :DINT;
END_VAR
END_METHOD

(*

## Short summary
This property returns the current state of the cycle manager according to its step.

.. <legal notes>

legal notes
=================
| SPDX-FileCopyrightText: © 2024 ekvip automation GmbH <info@ekvip.de>
| SPDX-License-Identifier: Apache-2.0
| For details check: Apache-2.0_

.. _Apache-2.0: https://www.apache.org/licenses/LICENSE-2.0

.. </legal notes>

*)
PROPERTY state :CNM_ReturnTypes.SingleExecutionState
GET
END_GET
END_PROPERTY

(*

## Short summary
This property returns the current, next and last step of the cycle manager via fluent interface with the ``ICycleSteps`` interfaces

.. <legal notes>

legal notes
=================
| SPDX-FileCopyrightText: © 2024 ekvip automation GmbH <info@ekvip.de>
| SPDX-License-Identifier: Apache-2.0
| For details check: Apache-2.0_

.. _Apache-2.0: https://www.apache.org/licenses/LICENSE-2.0

.. </legal notes>

*)
PROPERTY step :ICycleSteps
GET
END_GET
END_PROPERTY

(*

## Short summary
This method updates the current state and current step of the cycle manager. 
It needs to be called exactly once per PLC cycle per cycle manager instance.

.. <legal notes>

legal notes
=================
| SPDX-FileCopyrightText: © 2025 ekvip automation GmbH <info@ekvip.de>
| SPDX-License-Identifier: Apache-2.0
| For details check: Apache-2.0_

.. _Apache-2.0: https://www.apache.org/licenses/LICENSE-2.0

.. </legal notes>

*)


METHOD update
VAR_INPUT
	(*control bit to start or abort the cycle manager*)
	execute :BOOL;
	(*used for StopRequest evaluation if configured*)
	stopRequest :BOOL := FALSE;
	(*if true and Pausing Enabled and busy will proceed with PAUSE*)
	pause :BOOL := FALSE;
	(*if true, will acknowledge error and return to previous step*)
	resume :BOOL := FALSE;
	(* must be TRUE if stepping is enabled to proceed steps automatically *)
	stepControl :BOOL := TRUE;
END_VAR
END_METHOD

(*

## Short summary
This method waits for a boolean signal until the step can be changed. 

.. <legal notes>

legal notes
=================
| SPDX-FileCopyrightText: © 2024 ekvip automation GmbH <info@ekvip.de>
| SPDX-License-Identifier: Apache-2.0
| For details check: Apache-2.0_

.. _Apache-2.0: https://www.apache.org/licenses/LICENSE-2.0

.. </legal notes>

*)
METHOD waitFor
VAR_INPUT
	(* the value to wait for *)
	value :BOOL;
END_VAR
END_METHOD

END_INTERFACE

// ---- Project Information/F_GetCompany.TcPOU
// This function has been automatically generated from the project information.
{attribute 'signature_flag' := '1073741824'}
{attribute 'TcGenerated'}
{attribute 'no-analysis'}
FUNCTION F_GetCompany : WSTRING
VAR_INPUT
	
END_VAR

F_GetCompany := "ekvip automation GmbH";

END_FUNCTION

// ---- Project Information/F_GetTitle.TcPOU
// This function has been automatically generated from the project information.
{attribute 'signature_flag' := '1073741824'}
{attribute 'TcGenerated'}
{attribute 'no-analysis'}
FUNCTION F_GetTitle : WSTRING
VAR_INPUT
	
END_VAR

F_GetTitle := "CNM_CycleManagerInterfaces";

END_FUNCTION

// ---- Project Information/F_GetVersion.TcPOU
// This function has been automatically generated from the project information.
{attribute 'signature_flag' := '1073741824'}
{attribute 'TcGenerated'}
{attribute 'no-analysis'}
FUNCTION F_GetVersion : ST_LibVersion
VAR_INPUT
	
END_VAR

F_GetVersion.iMajor := 0;
F_GetVersion.iMinor := 1;
F_GetVersion.iBuild := 1;
F_GetVersion.iRevision := 0;
F_GetVersion.sVersion := '0.1.1.0';
F_GetVersion.nFlags := 0;

END_FUNCTION
